(* CODESYS project PLC.project

Project tree, tasks and I/O mapping:
  Device : CODESYS Control Win V3, 3S - Smart Software Solutions GmbH, version 3.5.3.50
    application Application
      libraries: Standard, 3.5.2.0 (System); Standard64, 3.5.2.0 (System); Util, 3.5.1.0 (System)
      task MainTask (cyclic, interval t#20ms, priority 1) calls unhappy_senario, sim, senario_happy, PLC_PRG, SIRINA_Programm, ON_OFF, LAMP_TESTING
      task VISU_TASK (cyclic, interval 100 ms, priority 30) calls VisuElems.Visu_Prg
      program PLC_PRG [SFC]: bcd, Silo_Visu, Init_Values, bcd_conveyor
      global variables GVL
      program ON_OFF [SFC]: CONTROL_OFF
      program SIRINA_Programm [SFC]: SET_WARNINGS, LIGHTS
      visualisation Visualization
      program LAMP_TESTING [SFC]: bcd, SET_VALUES
      program senario_happy [SFC]: Initial, Set_values, SET_values2, finish
      program unhappy_senario [SFC]: Initial, Set_values, SET_values2, ramp
      program sim [ST]
  text list GlobalTextList
  GlobalImagePool
  5ce3da45-db07-42e7-a21c-a00fff4ed8f6|5697-11187286.jpg
  5ce3da45-db07-42e7-a21c-a00fff4ed8f6|conveyor-belt-wheels-pack-vector-illustration-four-types-tracks-51926438.jpg
  5ce3da45-db07-42e7-a21c-a00fff4ed8f6|truck-icon-vectors_23-2147497003.jpg
  5ce3da45-db07-42e7-a21c-a00fff4ed8f6|apostol.jpg
  5ce3da45-db07-42e7-a21c-a00fff4ed8f6|frame.jpg
*)

// Device/Application/GVL
VAR_GLOBAL
	WRONG_SET_POINT_LIGHT: BOOL;
	SILO_EMPTY_LIGHT: BOOL;
	SIRINA: BOOL;
	VALVE_SILO: BOOL;
	MED_WEIGHT: INT;
	SILO_EMPTY: BOOL;
	VALVE_MED: BOOL;
	RUNNING: BOOL;
	ACKNOWLEDGE: BOOL;
	WRONG_SET_POINT: BOOL;
	BCD4: BYTE;
	BCD3: BYTE;
	BCD2: BYTE;
	// 	
	BCD1: BYTE;
	MED_MAX: INT;
	SET_POINT: INT;
	LOAD: BOOL;
	FILL: BOOL;
	TRUCK_ON_RAMP: BOOL;
	OFF: BOOL;
	ON: BOOL;
	SILO_WEIGHT: INT;
	CONTINUE_: BOOL;
	LAMP_TEST: BOOL;
	Senario: BOOL;
	TRASH_ON: BOOL;
	senario_un: BOOL;
END_VAR

// Device/Application/unhappy_senario
PROGRAM unhappy_senario

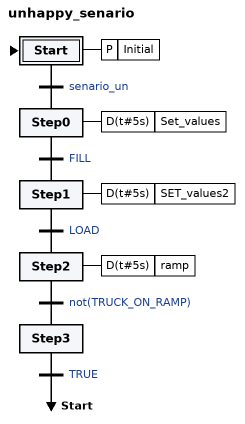
INITIAL_STEP Start:
    Initial(P);
END_STEP
TRANSITION FROM Start TO Step0
    := senario_un;
END_TRANSITION
STEP Step0:
    Set_values(D(t#5s));
END_STEP
TRANSITION FROM Step0 TO Step1
    := FILL;
END_TRANSITION
STEP Step1:
    SET_values2(D(t#5s));
END_STEP
TRANSITION FROM Step1 TO Step2
    := LOAD;
END_TRANSITION
STEP Step2:
    ramp(D(t#5s));
END_STEP
TRANSITION FROM Step2 TO Step3
    := not(TRUCK_ON_RAMP);
END_TRANSITION
STEP Step3:
END_STEP
TRANSITION FROM Step3 TO Start
    := TRUE;
END_TRANSITION

ACTION Initial:
senario_un := FALSE;
END_ACTION

ACTION Set_values:
ON := TRUE;
TRUCK_ON_RAMP := TRUE;
FILL := TRUE;
END_ACTION

ACTION SET_values2:
MED_WEIGHT := SET_POINT;
LOAD := TRUE;
END_ACTION

ACTION ramp:
TRUCK_ON_RAMP := FALSE;
END_ACTION

END_PROGRAM

// Device/Application/sim
PROGRAM sim
VAR
END_VAR

IF (VALVE_MED = TRUE) THEN
	TRASH_ON := TRUE;	
END_IF
IF (NOT(VALVE_MED OR RUNNING)) THEN
	TRASH_ON := FALSE;	
END_IF

END_PROGRAM

// Device/Application/senario_happy
PROGRAM senario_happy

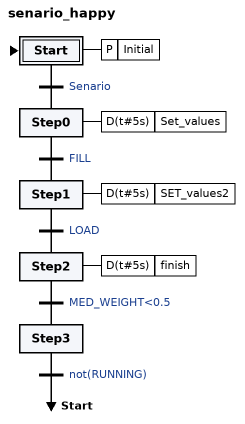
INITIAL_STEP Start:
    Initial(P);
END_STEP
TRANSITION FROM Start TO Step0
    := Senario;
END_TRANSITION
STEP Step0:
    Set_values(D(t#5s));
END_STEP
TRANSITION FROM Step0 TO Step1
    := FILL;
END_TRANSITION
STEP Step1:
    SET_values2(D(t#5s));
END_STEP
TRANSITION FROM Step1 TO Step2
    := LOAD;
END_TRANSITION
STEP Step2:
    finish(D(t#5s));
END_STEP
TRANSITION FROM Step2 TO Step3
    := MED_WEIGHT<0.5;
END_TRANSITION
STEP Step3:
END_STEP
TRANSITION FROM Step3 TO Start
    := not(RUNNING);
END_TRANSITION

ACTION Initial:
Senario := FALSE;
END_ACTION

ACTION Set_values:
ON := TRUE;
TRUCK_ON_RAMP := TRUE;
FILL := TRUE;
END_ACTION

ACTION SET_values2:
IF(MED_WEIGHT = SET_POINT) THEN
LOAD := TRUE;
END_IF
END_ACTION

ACTION finish:
MED_WEIGHT := 0;
END_ACTION

END_PROGRAM

// Device/Application/PLC_PRG
PROGRAM PLC_PRG
VAR
END_VAR

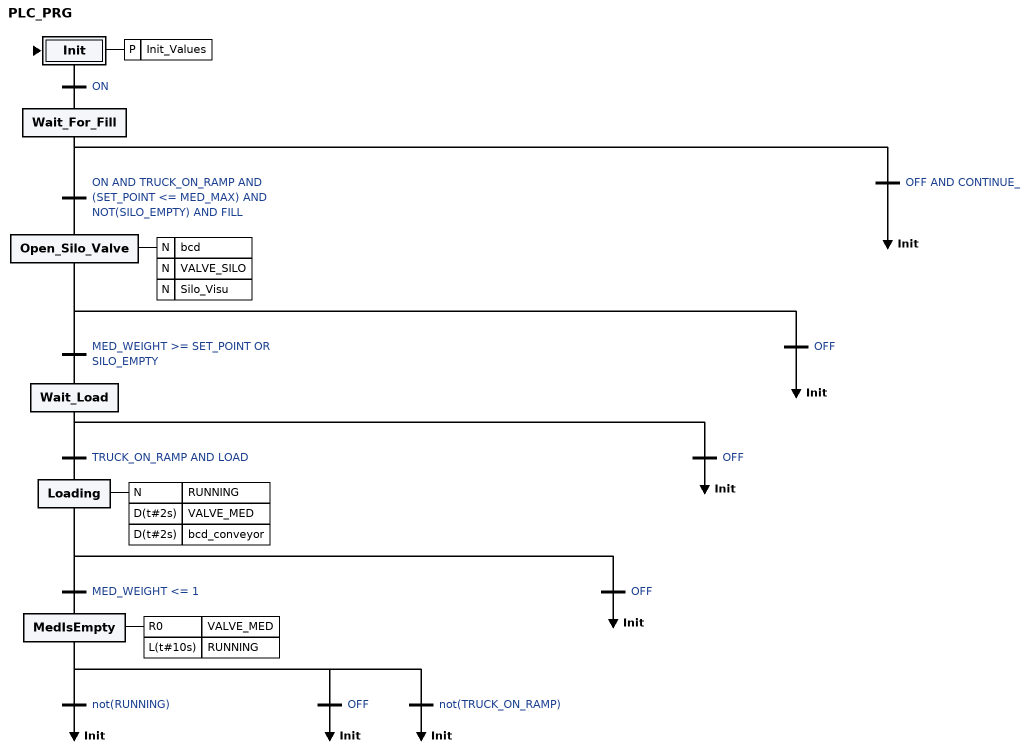
INITIAL_STEP Init:
    Init_Values(P);
END_STEP
TRANSITION FROM Init TO Wait_For_Fill
    := ON;
END_TRANSITION
STEP Wait_For_Fill:
END_STEP
TRANSITION FROM Wait_For_Fill TO Open_Silo_Valve
    := ON AND TRUCK_ON_RAMP AND (SET_POINT <= MED_MAX) AND NOT(SILO_EMPTY) AND FILL;
END_TRANSITION
TRANSITION FROM Wait_For_Fill TO Init
    := OFF AND CONTINUE_;
END_TRANSITION
STEP Open_Silo_Valve:
    bcd(N);
    VALVE_SILO(N);
    Silo_Visu(N);
END_STEP
TRANSITION FROM Open_Silo_Valve TO Wait_Load
    := MED_WEIGHT >= SET_POINT OR SILO_EMPTY;
END_TRANSITION
TRANSITION FROM Open_Silo_Valve TO Init
    := OFF;
END_TRANSITION
STEP Wait_Load:
END_STEP
TRANSITION FROM Wait_Load TO Loading
    := TRUCK_ON_RAMP AND LOAD;
END_TRANSITION
TRANSITION FROM Wait_Load TO Init
    := OFF;
END_TRANSITION
STEP Loading:
    RUNNING(N);
    VALVE_MED(D(t#2s));
    bcd_conveyor(D(t#2s));
END_STEP
TRANSITION FROM Loading TO MedIsEmpty
    := MED_WEIGHT <= 1;
END_TRANSITION
STEP MedIsEmpty:
    VALVE_MED(R0);
    RUNNING(L(t#10s));
END_STEP
TRANSITION FROM MedIsEmpty TO Init
    := not(RUNNING);
END_TRANSITION
TRANSITION FROM MedIsEmpty TO Init
    := OFF;
END_TRANSITION
TRANSITION FROM MedIsEmpty TO Init
    := not(TRUCK_ON_RAMP);
END_TRANSITION
TRANSITION FROM Loading TO Init
    := OFF;
END_TRANSITION

ACTION bcd:
SILO_WEIGHT := SILO_WEIGHT - 1;


//BCD ADD 1
BCD4 := BCD4 + 1 ;
IF (BCD4 = 10) THEN
	BCD4 := 0;
	BCD3 := BCD3 + 1;
	IF (BCD3 = 10) THEN
		BCD3 := 0;
		BCD2 := BCD2 + 1;
		IF (BCD2 = 10) THEN
			BCD2 := 0;
			BCD1 :=  BCD1 + 1;
		END_IF
	END_IF
END_IF

//BCD to INT
MED_WEIGHT := BCD1*1000 + BCD2*100 + BCD3*10 + BCD4 ;
END_ACTION

ACTION Silo_Visu:
SILO_WEIGHT := 5000;

IF (SILO_EMPTY) THEN
	SILO_WEIGHT := 0;
END_IF

SILO_WEIGHT := SILO_WEIGHT - MED_WEIGHT;
END_ACTION

ACTION Init_Values:
valve_silo := FALSE;
SIRINA := FALSE;
MED_WEIGHT := 0;
SILO_EMPTY := FALSE;
VALVE_MED := FALSE;
RUNNING := FALSE;
ACKNOWLEDGE := FALSE;
WRONG_SET_POINT := FALSE;
MED_MAX := 10000;
SET_POINT := 800;
LOAD := FALSE;
FILL := FALSE;
TRUCK_ON_RAMP := FALSE;
SILO_WEIGHT := 5000;
ON := FALSE;
OFF := TRUE;
CONTINUE_ := FALSE;
LAMP_TEST := FALSE;
END_ACTION

ACTION bcd_conveyor:

IF ( BCD4 = 0 ) THEN
	BCD4 := 9;
	IF (BCD3 = 0) THEN
		BCD3 := 9;
		IF (BCD2 = 0) THEN
			BCD2 := 9;
			//Don't check for overflow
			BCD1 := BCD1 - 1;
		ELSE
			BCD2 := BCD2 - 1;
		END_IF
	ELSE
		BCD3 := BCD3 - 1;
	END_IF
ELSE
	BCD4 := BCD4 - 1;
END_IF


//BCD TO INT
MED_WEIGHT := BCD1*1000 + BCD2*100 + BCD3*10 + BCD4 ;
END_ACTION

END_PROGRAM

// Device/Application/SIRINA_Programm
PROGRAM SIRINA_Programm
VAR
	BLINKER_WRONGsetPOINT: BLINK;
	BLINKER_SILOempty: BLINK;
END_VAR

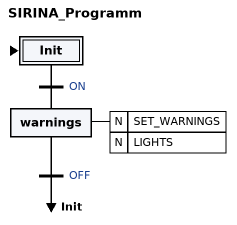
INITIAL_STEP Init:
END_STEP
TRANSITION FROM Init TO warnings
    := ON;
END_TRANSITION
STEP warnings:
    SET_WARNINGS(N);
    LIGHTS(N);
END_STEP
TRANSITION FROM warnings TO Init
    := OFF;
END_TRANSITION

ACTION SET_WARNINGS:
IF(SET_POINT > MED_MAX)THEN
	WRONG_SET_POINT := TRUE;
	IF(NOT(ACKNOWLEDGE))THEN
		SIRINA :=TRUE;
	END_IF
END_IF

IF(SILO_EMPTY AND NOT(ACKNOWLEDGE))THEN
	SIRINA := TRUE;
END_IF

IF(SET_POINT <= MED_MAX )THEN
	WRONG_SET_POINT := FALSE;
	IF(NOT(SILO_EMPTY))THEN
		SIRINA :=FALSE;
	END_IF
END_IF

IF(ACKNOWLEDGE)THEN
	SIRINA := FALSE;
END_IF
END_ACTION

ACTION LIGHTS:
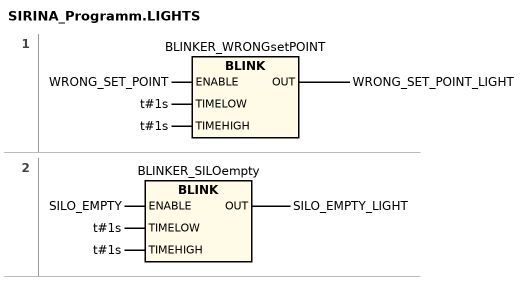
// NETWORK 1
BLINKER_WRONGsetPOINT(ENABLE := WRONG_SET_POINT, TIMELOW := t#1s, TIMEHIGH := t#1s); // BLINK
WRONG_SET_POINT_LIGHT := BLINKER_WRONGsetPOINT.OUT;

// NETWORK 2
BLINKER_SILOempty(ENABLE := SILO_EMPTY, TIMELOW := t#1s, TIMEHIGH := t#1s); // BLINK
SILO_EMPTY_LIGHT := BLINKER_SILOempty.OUT;
END_ACTION

END_PROGRAM

// Device/Application/ON_OFF
PROGRAM ON_OFF
VAR
END_VAR

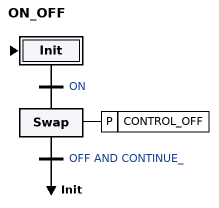
INITIAL_STEP Init:
END_STEP
TRANSITION FROM Init TO Swap
    := ON;
END_TRANSITION
STEP Swap:
    CONTROL_OFF(P);
END_STEP
TRANSITION FROM Swap TO Init
    := OFF AND CONTINUE_;
END_TRANSITION

ACTION CONTROL_OFF:
OFF := FALSE;
Continue_ := TRUE;
END_ACTION

END_PROGRAM

// Device/Application/LAMP_TESTING
PROGRAM LAMP_TESTING
VAR
END_VAR

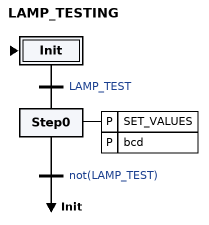
INITIAL_STEP Init:
END_STEP
TRANSITION FROM Init TO Step0
    := LAMP_TEST;
END_TRANSITION
STEP Step0:
    SET_VALUES(P);
    bcd(P);
END_STEP
TRANSITION FROM Step0 TO Init
    := not(LAMP_TEST);
END_TRANSITION

ACTION bcd:
SILO_WEIGHT := SILO_WEIGHT - 1;



BCD4 := BCD4 + 1 ;
IF (BCD4 = 10) THEN
	BCD4 := 0;
	BCD3 := BCD3 + 1;
	IF (BCD3 = 10) THEN
		BCD3 := 0;
		BCD2 := BCD2 + 1;
		IF (BCD2 = 10) THEN
			BCD2 := 0;
			BCD1 :=  BCD1 + 1;
		END_IF
	END_IF
END_IF


MED_WEIGHT := BCD1*1000 + BCD2*100 + BCD3*10 + BCD4 ;
END_ACTION

ACTION SET_VALUES:
ON := TRUE;
TRUCK_ON_RAMP := TRUE;
SILO_EMPTY := TRUE;
SET_POINT := MED_MAX+1;
BCD1 :=7;
BCD2 :=8;
BCD3 :=4;
BCD4 :=2;
END_ACTION

END_PROGRAM

// Device/Application/Visualization
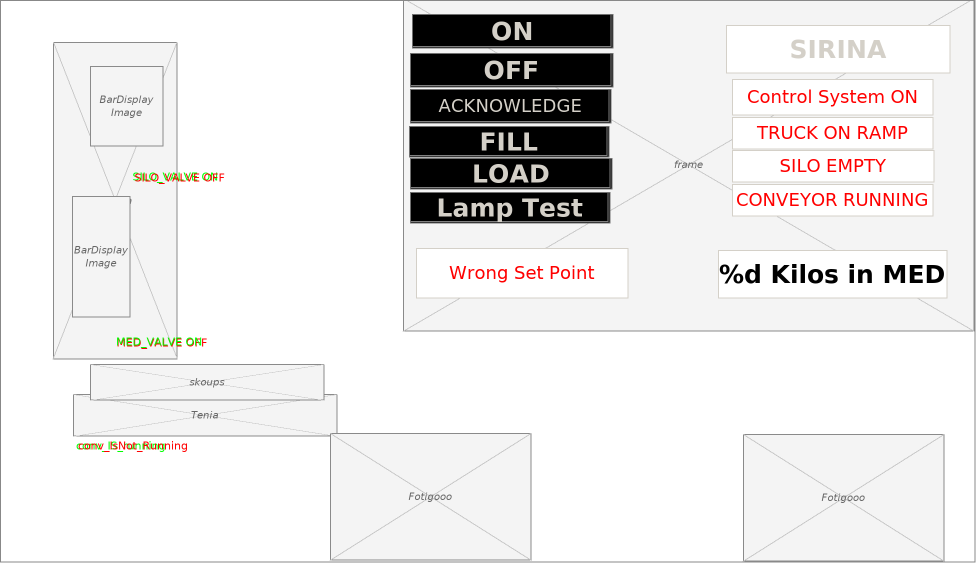
VISUALIZATION Visualization  // 976x563
    Image (403,-2 571x333), image: frame
    Textfield (416,248 212x50), "%d kilos", text variable: SET_POINT, invisible if: WRONG_SET_POINT
    Image (53,42 124x317), image: Doxeia
    Image (73,394 264x42), image: Tenia
    Image (743,434 201x127), invisible if: TRUCK_ON_RAMP, image: Fotigooo
    Image (330,433 201x127), invisible if: not(TRUCK_ON_RAMP), image: Fotigooo
    Image (90,364 234x36), invisible if: not(TRASH_ON), image: skoups
    Button (412,14 201x34), "ON", colour toggle: ON
        toggle ON p2164770859=TRUE
    Button (410,53 203x34), "OFF", colour toggle: OFF, pressed state: OFF
        OnMouseDown:  ToggleVariable=OFF
    Button (410,89 201x34), "ACKNOWLEDGE", colour toggle: ACKNOWLEDGE
        toggle ACKNOWLEDGE p2164770859=TRUE
    Button (409,126 200x31), "FILL", colour toggle: FILL, pressed state: FILL
        toggle FILL p2164770859=TRUE
    Button (410,158 202x31), "LOAD", colour toggle: LOAD, pressed state: LOAD
        toggle LOAD p2164770859=TRUE
    Button (410,192 200x31), "Lamp Test", colour toggle: LAMP_TEST, pressed state: LAMP_TEST
        toggle LAMP_TEST p2164770859=TRUE
    Textfield (416,248 212x50), "Wrong Set Point", colour toggle: WRONG_SET_POINT_LIGHT, invisible if: not(WRONG_SET_POINT)
    Textfield (718,250 229x48), "%d Kilos in MED", text variable: MED_WEIGHT
    Textfield (732,184 201x32), "CONVEYOR RUNNING", colour toggle: RUNNING, colour variable: 16777215
    Textfield (732,150 202x32), "SILO EMPTY", colour toggle: SILO_EMPTY_LIGHT, colour variable: 16777215
    Textfield (732,117 201x32), "TRUCK ON RAMP", colour toggle: TRUCK_ON_RAMP, colour variable: 16777215
    Textfield (732,79 201x36), "Control System ON", colour toggle: ON, colour variable: 16777215
    Textfield (726,25 224x48), "SIRINA", colour toggle: SIRINA, colour variable: 16777215
    Label (126,160 99x34), "SILO_VALVE ON", invisible if: not(VALVE_SILO)
    Label (105,163 150x30), "SILO_VALVE OFF", invisible if: VALVE_SILO
    Label (87,328 150x30), "MED_VALVE OFF", invisible if: VALVE_MED
    Label (84,327 150x30), "MED_VALVE ON", invisible if: not(VALVE_MED)
    Label (46,431 150x30), "conv_IS_running", invisible if: not(RUNNING)
    Label (58,431 150x30), "conv_IsNot_Running", invisible if: RUNNING
    BarDisplayImage (90,66 73x80), value: SILO_WEIGHT, style: BarDisplayImage-Gray, scale format: %.1f, scale 0..10000
    BarDisplayImage (72,196 58x121), value: MED_WEIGHT, style: BarDisplayImage-Gray, scale format: %.1f, scale 0..4000
END_VISUALIZATION
